(* CODESYS project Project_demo_2026_IOoff_v2_-_Codesys_SP20 (1)_RECOVERED_2026-05-21T15-52-03.project

Project tree, tasks and I/O mapping:
  Device : CODESYS Control Win V3 x64, CODESYS, version 3.5.20.40
    application Application
      libraries: Standard, 3.5.18.0 (System)
      task MainTask (cyclic, interval t#20ms, priority 1) calls PLC_PRG, SCADA_PRG, PRG_Loader, Order_generator
      function block Linear_Conveyor [SFC]: FB_Init, Receive_Workpiece_Data
      program PLC_PRG [CFC]
      data type Conv2Conv_bwd_T
      program Order_generator [ST]
      function block Cell [CFC]: FB_Init
      global variables GVL
      data type Conv2Conv_fwd_T
      data type Workpiece_T
      function block Machine_Conveyor [SFC]: FB_Init, Receive_Workpiece_Data, Inc_Next_Oper, Do_Change_Tool, Update_Tool, Copy_Next_Oper
      Symbols
      function block WarehouseIn_Conveyor [SFC]: Warehouse_Store_Piece, FB_Init, Warehouse_Rst_Piece, Receive_Workpiece_Data
      function block WarehouseOut_Conveyor [SFC]: FB_Init, Receive_Workpiece_Data, Warehouse_Req_Piece, Warehouse_Rst_Piece
      program SCADA_PRG [ST]
      data type Operation_T
      function block fb_Loader [ST]
      program PRG_Loader [ST]
      function block Transfer_Cell [CFC]: FB_Init
    Ethernet : Ethernet, CODESYS, version 4.2.0.0
      ModbusTCP_Slave_Device : ModbusTCP Server Device, CODESYS, version 4.4.0.0
          settings: UpdateableHolding = TRUE; DistinctBitAreas = TRUE; Coils Size = 8; Discrete Inputs Size = 8
          output S_sensor1 : BOOL  // Holding Registers.Holding Registers.Bit0
          output S_sensor2 : BOOL  // Holding Registers.Holding Registers.Bit1
          output S_sensor3 : BOOL  // Holding Registers.Holding Registers.Bit2
          output C1_stop : BOOL  // Holding Registers.Holding Registers.Bit0
          output C2_stop : BOOL  // Holding Registers.Holding Registers.Bit1
          output C3_stop : BOOL  // Holding Registers.Holding Registers.Bit2
          output Gate0 : BOOL  // Coils.Coils.Bit0
          output Gate1 : BOOL  // Coils.Coils.Bit1
          output Gate2 : BOOL  // Coils.Coils.Bit2
          unmapped channels: Holding Registers, Input Registers, Coils, Discrete Inputs
      Modbus_TCP_Master : Modbus TCP Client, CODESYS, version 4.4.0.0
          settings: AutoReconnect = TRUE
        Modbus_TCP_Slave : Modbus TCP Server, CODESYS, version 4.4.0.0
            settings: Unit-ID = 255; IPAddress = [127, 0, 0, 1]; Port = 5502; Channel 0.Function Code = 2; Channel 0.Read Offset = 16#0000; Channel 0.Read Length = 140; Channel 0.Write Offset = 0; Channel 0.Write Length = 0; Channel 0.Cycle Time = 100; Channel 1.Function Code = 15; Channel 1.Read Offset = 0; Channel 1.Read Length = 0; Channel 1.Write Offset = 16#0000; Channel 1.Write Length = 216; Channel 1.Cycle Time = 100; Channel 2.Function Code = 16; Channel 2.Read Offset = 0; Channel 2.Read Length = 0; Channel 2.Write Offset = 16#0000; Channel 2.Write Length = 15; Channel 2.Cycle Time = 100
            input  Application.GVL.In[0] : BOOL  // Channel 0.Channel 0.Bit0
            input  Application.GVL.In[1] : BOOL  // Channel 0.Channel 0.Bit1
            input  Application.GVL.In[2] : BOOL  // Channel 0.Channel 0.Bit2
            input  Application.GVL.In[3] : BOOL  // Channel 0.Channel 0.Bit3
            input  Application.GVL.In[4] : BOOL  // Channel 0.Channel 0.Bit4
            input  Application.GVL.In[5] : BOOL  // Channel 0.Channel 0.Bit5
            input  Application.GVL.In[6] : BOOL  // Channel 0.Channel 0.Bit6
            input  Application.GVL.In[7] : BOOL  // Channel 0.Channel 0.Bit7
            input  Application.GVL.In[8] : BOOL  // Channel 0.Channel 0.Bit0
            input  Application.GVL.In[9] : BOOL  // Channel 0.Channel 0.Bit1
            input  Application.GVL.In[10] : BOOL  // Channel 0.Channel 0.Bit2
            input  Application.GVL.In[11] : BOOL  // Channel 0.Channel 0.Bit3
            input  Application.GVL.In[12] : BOOL  // Channel 0.Channel 0.Bit4
            input  Application.GVL.In[13] : BOOL  // Channel 0.Channel 0.Bit5
            input  Application.GVL.In[14] : BOOL  // Channel 0.Channel 0.Bit6
            input  Application.GVL.In[15] : BOOL  // Channel 0.Channel 0.Bit7
            input  Application.GVL.In[16] : BOOL  // Channel 0.Channel 0.Bit0
            input  Application.GVL.In[17] : BOOL  // Channel 0.Channel 0.Bit1
            input  Application.GVL.In[18] : BOOL  // Channel 0.Channel 0.Bit2
            input  Application.GVL.In[19] : BOOL  // Channel 0.Channel 0.Bit3
            input  Application.GVL.In[20] : BOOL  // Channel 0.Channel 0.Bit4
            input  Application.GVL.In[21] : BOOL  // Channel 0.Channel 0.Bit5
            input  Application.GVL.In[22] : BOOL  // Channel 0.Channel 0.Bit6
            input  Application.GVL.In[23] : BOOL  // Channel 0.Channel 0.Bit7
            input  Application.GVL.In[24] : BOOL  // Channel 0.Channel 0.Bit0
            input  Application.GVL.In[25] : BOOL  // Channel 0.Channel 0.Bit1
            input  Application.GVL.In[26] : BOOL  // Channel 0.Channel 0.Bit2
            input  Application.GVL.In[27] : BOOL  // Channel 0.Channel 0.Bit3
            input  Application.GVL.In[28] : BOOL  // Channel 0.Channel 0.Bit4
            input  Application.GVL.In[29] : BOOL  // Channel 0.Channel 0.Bit5
            input  Application.GVL.In[30] : BOOL  // Channel 0.Channel 0.Bit6
            input  Application.GVL.In[31] : BOOL  // Channel 0.Channel 0.Bit7
            input  Application.GVL.In[32] : BOOL  // Channel 0.Channel 0.Bit0
            input  Application.GVL.In[33] : BOOL  // Channel 0.Channel 0.Bit1
            input  Application.GVL.In[34] : BOOL  // Channel 0.Channel 0.Bit2
            input  Application.GVL.In[35] : BOOL  // Channel 0.Channel 0.Bit3
            input  Application.GVL.In[36] : BOOL  // Channel 0.Channel 0.Bit4
            input  Application.GVL.In[37] : BOOL  // Channel 0.Channel 0.Bit5
            input  Application.GVL.In[38] : BOOL  // Channel 0.Channel 0.Bit6
            input  Application.GVL.In[39] : BOOL  // Channel 0.Channel 0.Bit7
            input  Application.GVL.In[40] : BOOL  // Channel 0.Channel 0.Bit0
            input  Application.GVL.In[41] : BOOL  // Channel 0.Channel 0.Bit1
            input  Application.GVL.In[42] : BOOL  // Channel 0.Channel 0.Bit2
            input  Application.GVL.In[43] : BOOL  // Channel 0.Channel 0.Bit3
            input  Application.GVL.In[44] : BOOL  // Channel 0.Channel 0.Bit4
            input  Application.GVL.In[45] : BOOL  // Channel 0.Channel 0.Bit5
            input  Application.GVL.In[46] : BOOL  // Channel 0.Channel 0.Bit6
            input  Application.GVL.In[47] : BOOL  // Channel 0.Channel 0.Bit7
            input  Application.GVL.In[48] : BOOL  // Channel 0.Channel 0.Bit0
            input  Application.GVL.In[49] : BOOL  // Channel 0.Channel 0.Bit1
            input  Application.GVL.In[50] : BOOL  // Channel 0.Channel 0.Bit2
            input  Application.GVL.In[51] : BOOL  // Channel 0.Channel 0.Bit3
            input  Application.GVL.In[52] : BOOL  // Channel 0.Channel 0.Bit4
            input  Application.GVL.In[53] : BOOL  // Channel 0.Channel 0.Bit5
            input  Application.GVL.In[54] : BOOL  // Channel 0.Channel 0.Bit6
            input  Application.GVL.In[55] : BOOL  // Channel 0.Channel 0.Bit7
            input  Application.GVL.In[56] : BOOL  // Channel 0.Channel 0.Bit0
            input  Application.GVL.In[57] : BOOL  // Channel 0.Channel 0.Bit1
            input  Application.GVL.In[58] : BOOL  // Channel 0.Channel 0.Bit2
            input  Application.GVL.In[59] : BOOL  // Channel 0.Channel 0.Bit3
            input  Application.GVL.In[60] : BOOL  // Channel 0.Channel 0.Bit4
            input  Application.GVL.In[61] : BOOL  // Channel 0.Channel 0.Bit5
            input  Application.GVL.In[62] : BOOL  // Channel 0.Channel 0.Bit6
            input  Application.GVL.In[63] : BOOL  // Channel 0.Channel 0.Bit7
            input  Application.GVL.In[64] : BOOL  // Channel 0.Channel 0.Bit0
            input  Application.GVL.In[65] : BOOL  // Channel 0.Channel 0.Bit1
            input  Application.GVL.In[66] : BOOL  // Channel 0.Channel 0.Bit2
            input  Application.GVL.In[67] : BOOL  // Channel 0.Channel 0.Bit3
            input  Application.GVL.In[68] : BOOL  // Channel 0.Channel 0.Bit4
            input  Application.GVL.In[69] : BOOL  // Channel 0.Channel 0.Bit5
            input  Application.GVL.In[70] : BOOL  // Channel 0.Channel 0.Bit6
            input  Application.GVL.In[71] : BOOL  // Channel 0.Channel 0.Bit7
            input  Application.GVL.In[72] : BOOL  // Channel 0.Channel 0.Bit0
            input  Application.GVL.In[73] : BOOL  // Channel 0.Channel 0.Bit1
            input  Application.GVL.In[74] : BOOL  // Channel 0.Channel 0.Bit2
            input  Application.GVL.In[75] : BOOL  // Channel 0.Channel 0.Bit3
            input  Application.GVL.In[76] : BOOL  // Channel 0.Channel 0.Bit4
            input  Application.GVL.In[77] : BOOL  // Channel 0.Channel 0.Bit5
            input  Application.GVL.In[78] : BOOL  // Channel 0.Channel 0.Bit6
            input  Application.GVL.In[79] : BOOL  // Channel 0.Channel 0.Bit7
            input  Application.GVL.In[80] : BOOL  // Channel 0.Channel 0.Bit0
            input  Application.GVL.In[81] : BOOL  // Channel 0.Channel 0.Bit1
            input  Application.GVL.In[82] : BOOL  // Channel 0.Channel 0.Bit2
            input  Application.GVL.In[83] : BOOL  // Channel 0.Channel 0.Bit3
            input  Application.GVL.In[84] : BOOL  // Channel 0.Channel 0.Bit4
            input  Application.GVL.In[85] : BOOL  // Channel 0.Channel 0.Bit5
            input  Application.GVL.In[86] : BOOL  // Channel 0.Channel 0.Bit6
            input  Application.GVL.In[87] : BOOL  // Channel 0.Channel 0.Bit7
            input  Application.GVL.In[88] : BOOL  // Channel 0.Channel 0.Bit0
            input  Application.GVL.In[89] : BOOL  // Channel 0.Channel 0.Bit1
            input  Application.GVL.In[90] : BOOL  // Channel 0.Channel 0.Bit2
            input  Application.GVL.In[91] : BOOL  // Channel 0.Channel 0.Bit3
            input  Application.GVL.In[92] : BOOL  // Channel 0.Channel 0.Bit4
            input  Application.GVL.In[93] : BOOL  // Channel 0.Channel 0.Bit5
            input  Application.GVL.In[94] : BOOL  // Channel 0.Channel 0.Bit6
            input  Application.GVL.In[95] : BOOL  // Channel 0.Channel 0.Bit7
            input  Application.GVL.In[96] : BOOL  // Channel 0.Channel 0.Bit0
            input  Application.GVL.In[97] : BOOL  // Channel 0.Channel 0.Bit1
            input  Application.GVL.In[98] : BOOL  // Channel 0.Channel 0.Bit2
            input  Application.GVL.In[99] : BOOL  // Channel 0.Channel 0.Bit3
            input  Application.GVL.In[100] : BOOL  // Channel 0.Channel 0.Bit4
            input  Application.GVL.In[101] : BOOL  // Channel 0.Channel 0.Bit5
            input  Application.GVL.In[102] : BOOL  // Channel 0.Channel 0.Bit6
            input  Application.GVL.In[103] : BOOL  // Channel 0.Channel 0.Bit7
            input  Application.GVL.In[104] : BOOL  // Channel 0.Channel 0.Bit0
            input  Application.GVL.In[105] : BOOL  // Channel 0.Channel 0.Bit1
            input  Application.GVL.In[106] : BOOL  // Channel 0.Channel 0.Bit2
            input  Application.GVL.In[107] : BOOL  // Channel 0.Channel 0.Bit3
            input  Application.GVL.In[108] : BOOL  // Channel 0.Channel 0.Bit4
            input  Application.GVL.In[109] : BOOL  // Channel 0.Channel 0.Bit5
            input  Application.GVL.In[110] : BOOL  // Channel 0.Channel 0.Bit6
            input  Application.GVL.In[111] : BOOL  // Channel 0.Channel 0.Bit7
            input  Application.GVL.In[112] : BOOL  // Channel 0.Channel 0.Bit0
            input  Application.GVL.In[113] : BOOL  // Channel 0.Channel 0.Bit1
            input  Application.GVL.In[114] : BOOL  // Channel 0.Channel 0.Bit2
            input  Application.GVL.In[115] : BOOL  // Channel 0.Channel 0.Bit3
            input  Application.GVL.In[116] : BOOL  // Channel 0.Channel 0.Bit4
            input  Application.GVL.In[117] : BOOL  // Channel 0.Channel 0.Bit5
            input  Application.GVL.In[118] : BOOL  // Channel 0.Channel 0.Bit6
            input  Application.GVL.In[119] : BOOL  // Channel 0.Channel 0.Bit7
            input  Application.GVL.In[120] : BOOL  // Channel 0.Channel 0.Bit0
            input  Application.GVL.In[121] : BOOL  // Channel 0.Channel 0.Bit1
            input  Application.GVL.In[122] : BOOL  // Channel 0.Channel 0.Bit2
            input  Application.GVL.In[123] : BOOL  // Channel 0.Channel 0.Bit3
            input  Application.GVL.In[124] : BOOL  // Channel 0.Channel 0.Bit4
            input  Application.GVL.In[125] : BOOL  // Channel 0.Channel 0.Bit5
            input  Application.GVL.In[126] : BOOL  // Channel 0.Channel 0.Bit6
            input  Application.GVL.In[127] : BOOL  // Channel 0.Channel 0.Bit7
            input  Application.GVL.In[128] : BOOL  // Channel 0.Channel 0.Bit0
            input  Application.GVL.In[129] : BOOL  // Channel 0.Channel 0.Bit1
            input  Application.GVL.In[130] : BOOL  // Channel 0.Channel 0.Bit2
            input  Application.GVL.In[131] : BOOL  // Channel 0.Channel 0.Bit3
            input  Application.GVL.In[132] : BOOL  // Channel 0.Channel 0.Bit4
            input  Application.GVL.In[133] : BOOL  // Channel 0.Channel 0.Bit5
            input  Application.GVL.In[134] : BOOL  // Channel 0.Channel 0.Bit6
            input  Application.GVL.In[135] : BOOL  // Channel 0.Channel 0.Bit7
            input  Application.GVL.In[136] : BOOL  // Channel 0.Channel 0.Bit0
            input  Application.GVL.In[137] : BOOL  // Channel 0.Channel 0.Bit1
            input  Application.GVL.In[138] : BOOL  // Channel 0.Channel 0.Bit2
            input  Application.GVL.In[139] : BOOL  // Channel 0.Channel 0.Bit3
            output Application.GVL.Out[0] : BOOL  // Channel 1.Channel 1.Bit0
            output Application.GVL.Out[1] : BOOL  // Channel 1.Channel 1.Bit1
            output Application.GVL.Out[2] : BOOL  // Channel 1.Channel 1.Bit2
            output Application.GVL.Out[3] : BOOL  // Channel 1.Channel 1.Bit3
            output Application.GVL.Out[4] : BOOL  // Channel 1.Channel 1.Bit4
            output Application.GVL.Out[5] : BOOL  // Channel 1.Channel 1.Bit5
            output Application.GVL.Out[6] : BOOL  // Channel 1.Channel 1.Bit6
            output Application.GVL.Out[7] : BOOL  // Channel 1.Channel 1.Bit7
            output Application.GVL.Out[8] : BOOL  // Channel 1.Channel 1.Bit0
            output Application.GVL.Out[9] : BOOL  // Channel 1.Channel 1.Bit1
            output Application.GVL.Out[10] : BOOL  // Channel 1.Channel 1.Bit2
            output Application.GVL.Out[11] : BOOL  // Channel 1.Channel 1.Bit3
            output Application.GVL.Out[12] : BOOL  // Channel 1.Channel 1.Bit4
            output Application.GVL.Out[13] : BOOL  // Channel 1.Channel 1.Bit5
            output Application.GVL.Out[14] : BOOL  // Channel 1.Channel 1.Bit6
            output Application.GVL.Out[15] : BOOL  // Channel 1.Channel 1.Bit7
            output Application.GVL.Out[16] : BOOL  // Channel 1.Channel 1.Bit0
            output Application.GVL.Out[17] : BOOL  // Channel 1.Channel 1.Bit1
            output Application.GVL.Out[18] : BOOL  // Channel 1.Channel 1.Bit2
            output Application.GVL.Out[19] : BOOL  // Channel 1.Channel 1.Bit3
            output Application.GVL.Out[20] : BOOL  // Channel 1.Channel 1.Bit4
            output Application.GVL.Out[21] : BOOL  // Channel 1.Channel 1.Bit5
            output Application.GVL.Out[22] : BOOL  // Channel 1.Channel 1.Bit6
            output Application.GVL.Out[23] : BOOL  // Channel 1.Channel 1.Bit7
            output Application.GVL.Out[24] : BOOL  // Channel 1.Channel 1.Bit0
            output Application.GVL.Out[25] : BOOL  // Channel 1.Channel 1.Bit1
            output Application.GVL.Out[26] : BOOL  // Channel 1.Channel 1.Bit2
            output Application.GVL.Out[27] : BOOL  // Channel 1.Channel 1.Bit3
            output Application.GVL.Out[28] : BOOL  // Channel 1.Channel 1.Bit4
            output Application.GVL.Out[29] : BOOL  // Channel 1.Channel 1.Bit5
            output Application.GVL.Out[30] : BOOL  // Channel 1.Channel 1.Bit6
            output Application.GVL.Out[31] : BOOL  // Channel 1.Channel 1.Bit7
            output Application.GVL.Out[32] : BOOL  // Channel 1.Channel 1.Bit0
            output Application.GVL.Out[33] : BOOL  // Channel 1.Channel 1.Bit1
            output Application.GVL.Out[34] : BOOL  // Channel 1.Channel 1.Bit2
            output Application.GVL.Out[35] : BOOL  // Channel 1.Channel 1.Bit3
            output Application.GVL.Out[36] : BOOL  // Channel 1.Channel 1.Bit4
            output Application.GVL.Out[37] : BOOL  // Channel 1.Channel 1.Bit5
            output Application.GVL.Out[38] : BOOL  // Channel 1.Channel 1.Bit6
            output Application.GVL.Out[39] : BOOL  // Channel 1.Channel 1.Bit7
            output Application.GVL.Out[40] : BOOL  // Channel 1.Channel 1.Bit0
            output Application.GVL.Out[41] : BOOL  // Channel 1.Channel 1.Bit1
            output Application.GVL.Out[42] : BOOL  // Channel 1.Channel 1.Bit2
            output Application.GVL.Out[43] : BOOL  // Channel 1.Channel 1.Bit3
            output Application.GVL.Out[44] : BOOL  // Channel 1.Channel 1.Bit4
            output Application.GVL.Out[45] : BOOL  // Channel 1.Channel 1.Bit5
            output Application.GVL.Out[46] : BOOL  // Channel 1.Channel 1.Bit6
            output Application.GVL.Out[47] : BOOL  // Channel 1.Channel 1.Bit7
            output Application.GVL.Out[48] : BOOL  // Channel 1.Channel 1.Bit0
            output Application.GVL.Out[49] : BOOL  // Channel 1.Channel 1.Bit1
            output Application.GVL.Out[50] : BOOL  // Channel 1.Channel 1.Bit2
            output Application.GVL.Out[51] : BOOL  // Channel 1.Channel 1.Bit3
            output Application.GVL.Out[52] : BOOL  // Channel 1.Channel 1.Bit4
            output Application.GVL.Out[53] : BOOL  // Channel 1.Channel 1.Bit5
            output Application.GVL.Out[54] : BOOL  // Channel 1.Channel 1.Bit6
            output Application.GVL.Out[55] : BOOL  // Channel 1.Channel 1.Bit7
            output Application.GVL.Out[56] : BOOL  // Channel 1.Channel 1.Bit0
            output Application.GVL.Out[57] : BOOL  // Channel 1.Channel 1.Bit1
            output Application.GVL.Out[58] : BOOL  // Channel 1.Channel 1.Bit2
            output Application.GVL.Out[59] : BOOL  // Channel 1.Channel 1.Bit3
            output Application.GVL.Out[60] : BOOL  // Channel 1.Channel 1.Bit4
            output Application.GVL.Out[61] : BOOL  // Channel 1.Channel 1.Bit5
            output Application.GVL.Out[62] : BOOL  // Channel 1.Channel 1.Bit6
            output Application.GVL.Out[63] : BOOL  // Channel 1.Channel 1.Bit7
            output Application.GVL.Out[64] : BOOL  // Channel 1.Channel 1.Bit0
            output Application.GVL.Out[65] : BOOL  // Channel 1.Channel 1.Bit1
            output Application.GVL.Out[66] : BOOL  // Channel 1.Channel 1.Bit2
            output Application.GVL.Out[67] : BOOL  // Channel 1.Channel 1.Bit3
            output Application.GVL.Out[68] : BOOL  // Channel 1.Channel 1.Bit4
            output Application.GVL.Out[69] : BOOL  // Channel 1.Channel 1.Bit5
            output Application.GVL.Out[70] : BOOL  // Channel 1.Channel 1.Bit6
            output Application.GVL.Out[71] : BOOL  // Channel 1.Channel 1.Bit7
            output Application.GVL.Out[72] : BOOL  // Channel 1.Channel 1.Bit0
            output Application.GVL.Out[73] : BOOL  // Channel 1.Channel 1.Bit1
            output Application.GVL.Out[74] : BOOL  // Channel 1.Channel 1.Bit2
            output Application.GVL.Out[75] : BOOL  // Channel 1.Channel 1.Bit3
            output Application.GVL.Out[76] : BOOL  // Channel 1.Channel 1.Bit4
            output Application.GVL.Out[77] : BOOL  // Channel 1.Channel 1.Bit5
            output Application.GVL.Out[78] : BOOL  // Channel 1.Channel 1.Bit6
            output Application.GVL.Out[79] : BOOL  // Channel 1.Channel 1.Bit7
            output Application.GVL.Out[80] : BOOL  // Channel 1.Channel 1.Bit0
            output Application.GVL.Out[81] : BOOL  // Channel 1.Channel 1.Bit1
            output Application.GVL.Out[82] : BOOL  // Channel 1.Channel 1.Bit2
            output Application.GVL.Out[83] : BOOL  // Channel 1.Channel 1.Bit3
            output Application.GVL.Out[84] : BOOL  // Channel 1.Channel 1.Bit4
            output Application.GVL.Out[85] : BOOL  // Channel 1.Channel 1.Bit5
            output Application.GVL.Out[86] : BOOL  // Channel 1.Channel 1.Bit6
            output Application.GVL.Out[87] : BOOL  // Channel 1.Channel 1.Bit7
            output Application.GVL.Out[88] : BOOL  // Channel 1.Channel 1.Bit0
            output Application.GVL.Out[89] : BOOL  // Channel 1.Channel 1.Bit1
            output Application.GVL.Out[90] : BOOL  // Channel 1.Channel 1.Bit2
            output Application.GVL.Out[91] : BOOL  // Channel 1.Channel 1.Bit3
            output Application.GVL.Out[92] : BOOL  // Channel 1.Channel 1.Bit4
            output Application.GVL.Out[93] : BOOL  // Channel 1.Channel 1.Bit5
            output Application.GVL.Out[94] : BOOL  // Channel 1.Channel 1.Bit6
            output Application.GVL.Out[95] : BOOL  // Channel 1.Channel 1.Bit7
            output Application.GVL.Out[96] : BOOL  // Channel 1.Channel 1.Bit0
            output Application.GVL.Out[97] : BOOL  // Channel 1.Channel 1.Bit1
            output Application.GVL.Out[98] : BOOL  // Channel 1.Channel 1.Bit2
            output Application.GVL.Out[99] : BOOL  // Channel 1.Channel 1.Bit3
            output Application.GVL.Out[100] : BOOL  // Channel 1.Channel 1.Bit4
            output Application.GVL.Out[101] : BOOL  // Channel 1.Channel 1.Bit5
            output Application.GVL.Out[102] : BOOL  // Channel 1.Channel 1.Bit6
            output Application.GVL.Out[103] : BOOL  // Channel 1.Channel 1.Bit7
            output Application.GVL.Out[104] : BOOL  // Channel 1.Channel 1.Bit0
            output Application.GVL.Out[105] : BOOL  // Channel 1.Channel 1.Bit1
            output Application.GVL.Out[106] : BOOL  // Channel 1.Channel 1.Bit2
            output Application.GVL.Out[107] : BOOL  // Channel 1.Channel 1.Bit3
            output Application.GVL.Out[108] : BOOL  // Channel 1.Channel 1.Bit4
            output Application.GVL.Out[109] : BOOL  // Channel 1.Channel 1.Bit5
            output Application.GVL.Out[110] : BOOL  // Channel 1.Channel 1.Bit6
            output Application.GVL.Out[111] : BOOL  // Channel 1.Channel 1.Bit7
            output Application.GVL.Out[112] : BOOL  // Channel 1.Channel 1.Bit0
            output Application.GVL.Out[113] : BOOL  // Channel 1.Channel 1.Bit1
            output Application.GVL.Out[114] : BOOL  // Channel 1.Channel 1.Bit2
            output Application.GVL.Out[115] : BOOL  // Channel 1.Channel 1.Bit3
            output Application.GVL.Out[116] : BOOL  // Channel 1.Channel 1.Bit4
            output Application.GVL.Out[117] : BOOL  // Channel 1.Channel 1.Bit5
            output Application.GVL.Out[118] : BOOL  // Channel 1.Channel 1.Bit6
            output Application.GVL.Out[119] : BOOL  // Channel 1.Channel 1.Bit7
            output Application.GVL.Out[120] : BOOL  // Channel 1.Channel 1.Bit0
            output Application.GVL.Out[121] : BOOL  // Channel 1.Channel 1.Bit1
            output Application.GVL.Out[122] : BOOL  // Channel 1.Channel 1.Bit2
            output Application.GVL.Out[123] : BOOL  // Channel 1.Channel 1.Bit3
            output Application.GVL.Out[124] : BOOL  // Channel 1.Channel 1.Bit4
            output Application.GVL.Out[125] : BOOL  // Channel 1.Channel 1.Bit5
            output Application.GVL.Out[126] : BOOL  // Channel 1.Channel 1.Bit6
            output Application.GVL.Out[127] : BOOL  // Channel 1.Channel 1.Bit7
            output Application.GVL.Out[128] : BOOL  // Channel 1.Channel 1.Bit0
            output Application.GVL.Out[129] : BOOL  // Channel 1.Channel 1.Bit1
            output Application.GVL.Out[130] : BOOL  // Channel 1.Channel 1.Bit2
            output Application.GVL.Out[131] : BOOL  // Channel 1.Channel 1.Bit3
            output Application.GVL.Out[132] : BOOL  // Channel 1.Channel 1.Bit4
            output Application.GVL.Out[133] : BOOL  // Channel 1.Channel 1.Bit5
            output Application.GVL.Out[134] : BOOL  // Channel 1.Channel 1.Bit6
            output Application.GVL.Out[135] : BOOL  // Channel 1.Channel 1.Bit7
            output Application.GVL.Out[136] : BOOL  // Channel 1.Channel 1.Bit0
            output Application.GVL.Out[137] : BOOL  // Channel 1.Channel 1.Bit1
            output Application.GVL.Out[138] : BOOL  // Channel 1.Channel 1.Bit2
            output Application.GVL.Out[139] : BOOL  // Channel 1.Channel 1.Bit3
            output Application.GVL.Out[140] : BOOL  // Channel 1.Channel 1.Bit4
            output Application.GVL.Out[141] : BOOL  // Channel 1.Channel 1.Bit5
            output Application.GVL.Out[142] : BOOL  // Channel 1.Channel 1.Bit6
            output Application.GVL.Out[143] : BOOL  // Channel 1.Channel 1.Bit7
            output Application.GVL.Out[144] : BOOL  // Channel 1.Channel 1.Bit0
            output Application.GVL.Out[145] : BOOL  // Channel 1.Channel 1.Bit1
            output Application.GVL.Out[146] : BOOL  // Channel 1.Channel 1.Bit2
            output Application.GVL.Out[147] : BOOL  // Channel 1.Channel 1.Bit3
            output Application.GVL.Out[148] : BOOL  // Channel 1.Channel 1.Bit4
            output Application.GVL.Out[149] : BOOL  // Channel 1.Channel 1.Bit5
            output Application.GVL.Out[150] : BOOL  // Channel 1.Channel 1.Bit6
            output Application.GVL.Out[151] : BOOL  // Channel 1.Channel 1.Bit7
            output Application.GVL.Out[152] : BOOL  // Channel 1.Channel 1.Bit0
            output Application.GVL.Out[153] : BOOL  // Channel 1.Channel 1.Bit1
            output Application.GVL.Out[154] : BOOL  // Channel 1.Channel 1.Bit2
            output Application.GVL.Out[155] : BOOL  // Channel 1.Channel 1.Bit3
            output Application.GVL.Out[156] : BOOL  // Channel 1.Channel 1.Bit4
            output Application.GVL.Out[157] : BOOL  // Channel 1.Channel 1.Bit5
            output Application.GVL.Out[158] : BOOL  // Channel 1.Channel 1.Bit6
            output Application.GVL.Out[159] : BOOL  // Channel 1.Channel 1.Bit7
            output Application.GVL.Out[160] : BOOL  // Channel 1.Channel 1.Bit0
            output Application.GVL.Out[161] : BOOL  // Channel 1.Channel 1.Bit1
            output Application.GVL.Out[162] : BOOL  // Channel 1.Channel 1.Bit2
            output Application.GVL.Out[163] : BOOL  // Channel 1.Channel 1.Bit3
            output Application.GVL.Out[164] : BOOL  // Channel 1.Channel 1.Bit4
            output Application.GVL.Out[165] : BOOL  // Channel 1.Channel 1.Bit5
            output Application.GVL.Out[166] : BOOL  // Channel 1.Channel 1.Bit6
            output Application.GVL.Out[167] : BOOL  // Channel 1.Channel 1.Bit7
            output Application.GVL.Out[168] : BOOL  // Channel 1.Channel 1.Bit0
            output Application.GVL.Out[169] : BOOL  // Channel 1.Channel 1.Bit1
            output Application.GVL.Out[170] : BOOL  // Channel 1.Channel 1.Bit2
            output Application.GVL.Out[171] : BOOL  // Channel 1.Channel 1.Bit3
            output Application.GVL.Out[172] : BOOL  // Channel 1.Channel 1.Bit4
            output Application.GVL.Out[173] : BOOL  // Channel 1.Channel 1.Bit5
            output Application.GVL.Out[174] : BOOL  // Channel 1.Channel 1.Bit6
            output Application.GVL.Out[175] : BOOL  // Channel 1.Channel 1.Bit7
            output Application.GVL.Out[176] : BOOL  // Channel 1.Channel 1.Bit0
            output Application.GVL.Out[177] : BOOL  // Channel 1.Channel 1.Bit1
            output Application.GVL.Out[178] : BOOL  // Channel 1.Channel 1.Bit2
            output Application.GVL.Out[179] : BOOL  // Channel 1.Channel 1.Bit3
            output Application.GVL.Out[180] : BOOL  // Channel 1.Channel 1.Bit4
            output Application.GVL.Out[181] : BOOL  // Channel 1.Channel 1.Bit5
            output Application.GVL.Out[182] : BOOL  // Channel 1.Channel 1.Bit6
            output Application.GVL.Out[183] : BOOL  // Channel 1.Channel 1.Bit7
            output Application.GVL.Out[184] : BOOL  // Channel 1.Channel 1.Bit0
            output Application.GVL.Out[185] : BOOL  // Channel 1.Channel 1.Bit1
            output Application.GVL.Out[186] : BOOL  // Channel 1.Channel 1.Bit2
            output Application.GVL.Out[187] : BOOL  // Channel 1.Channel 1.Bit3
            output Application.GVL.Out[188] : BOOL  // Channel 1.Channel 1.Bit4
            output Application.GVL.Out[189] : BOOL  // Channel 1.Channel 1.Bit5
            output Application.GVL.Out[190] : BOOL  // Channel 1.Channel 1.Bit6
            output Application.GVL.Out[191] : BOOL  // Channel 1.Channel 1.Bit7
            output Application.GVL.Out[192] : BOOL  // Channel 1.Channel 1.Bit0
            output Application.GVL.Out[193] : BOOL  // Channel 1.Channel 1.Bit1
            output Application.GVL.Out[194] : BOOL  // Channel 1.Channel 1.Bit2
            output Application.GVL.Out[195] : BOOL  // Channel 1.Channel 1.Bit3
            output Application.GVL.Out[196] : BOOL  // Channel 1.Channel 1.Bit4
            output Application.GVL.Out[197] : BOOL  // Channel 1.Channel 1.Bit5
            output Application.GVL.Out[198] : BOOL  // Channel 1.Channel 1.Bit6
            output Application.GVL.Out[199] : BOOL  // Channel 1.Channel 1.Bit7
            output Application.GVL.Out[200] : BOOL  // Channel 1.Channel 1.Bit0
            output Application.GVL.Out[201] : BOOL  // Channel 1.Channel 1.Bit1
            output Application.GVL.Out[202] : BOOL  // Channel 1.Channel 1.Bit2
            output Application.GVL.Out[203] : BOOL  // Channel 1.Channel 1.Bit3
            output Application.GVL.Out[204] : BOOL  // Channel 1.Channel 1.Bit4
            output Application.GVL.Out[205] : BOOL  // Channel 1.Channel 1.Bit5
            output Application.GVL.Out[206] : BOOL  // Channel 1.Channel 1.Bit6
            output Application.GVL.Out[207] : BOOL  // Channel 1.Channel 1.Bit7
            output Application.GVL.Out[208] : BOOL  // Channel 1.Channel 1.Bit0
            output Application.GVL.Out[209] : BOOL  // Channel 1.Channel 1.Bit1
            output Application.GVL.Out[210] : BOOL  // Channel 1.Channel 1.Bit2
            output Application.GVL.Out[211] : BOOL  // Channel 1.Channel 1.Bit3
            output Application.GVL.Out[212] : BOOL  // Channel 1.Channel 1.Bit4
            output Application.GVL.Out[213] : BOOL  // Channel 1.Channel 1.Bit5
            output Application.GVL.Out[214] : BOOL  // Channel 1.Channel 1.Bit6
            output Application.GVL.Out[215] : BOOL  // Channel 1.Channel 1.Bit7
            output Application.GVL.Reg[0] : WORD  // Channel 2.Channel 2
            output Application.GVL.Reg[1] : WORD  // Channel 2.Channel 2
            output Application.GVL.Reg[2] : WORD  // Channel 2.Channel 2
            output Application.GVL.Reg[3] : WORD  // Channel 2.Channel 2
            output Application.GVL.Reg[4] : WORD  // Channel 2.Channel 2
            output Application.GVL.Reg[5] : WORD  // Channel 2.Channel 2
            output Application.GVL.Reg[6] : WORD  // Channel 2.Channel 2
            output Application.GVL.Reg[7] : WORD  // Channel 2.Channel 2
            output Application.GVL.Reg[8] : WORD  // Channel 2.Channel 2
            output Application.GVL.Reg[9] : WORD  // Channel 2.Channel 2
            output Application.GVL.Reg[10] : WORD  // Channel 2.Channel 2
            output Application.GVL.Reg[11] : WORD  // Channel 2.Channel 2
            output Application.GVL.Reg[12] : WORD  // Channel 2.Channel 2
            output Application.GVL.Reg[13] : WORD  // Channel 2.Channel 2
            output Application.GVL.Reg[14] : WORD  // Channel 2.Channel 2
            unmapped channels: Channel 0, Channel 1, Channel 2
*)

// Device/Application/Conv2Conv_bwd_T
TYPE Conv2Conv_bwd_T :
STRUCT
		free_cmd: BOOL;
END_STRUCT
END_TYPE

// Device/Application/Conv2Conv_fwd_T
TYPE Conv2Conv_fwd_T :
STRUCT
		recv_cmd: BOOL;
		Workpiece: Workpiece_T;
END_STRUCT
END_TYPE

// Device/Application/Workpiece_T
TYPE Workpiece_T :
STRUCT
	InitPiece: INT;
	Operations: ARRAY [0 .. 10] OF Operation_T;
	Next_Operation: INT;
	Last_Operation: INT;
END_STRUCT
END_TYPE

// Device/Application/Operation_T
TYPE Operation_T :
STRUCT
	Cell: INT;
	Machine: INT;
	Tool: INT;
	OpTime: TIME;
END_STRUCT
END_TYPE

// Device/Application/GVL
{attribute 'qualified_only'}
VAR_GLOBAL
	In:  ARRAY [0 .. 139] OF BOOL;
	Out: ARRAY [0 .. 215] OF BOOL;
	Reg: ARRAY [0 .. 14] OF UINT;
	
	Cell_1_Top_Order:  Conv2conv_fwd_T;
	Cell_1_Top_Status: Conv2conv_bwd_T;
	
	Cell_2_Top_Order:  Conv2conv_fwd_T;
	Cell_2_Top_Status: Conv2conv_bwd_T;
	
	// Add to existing GVL VAR_GLOBAL block:

	// Cells 3 & 4 handshakes (já tens no PLC_PRG, move-os para GVL para acesso OPC-UA)
	Cell_3_Top_Order:  Conv2Conv_fwd_T;
	Cell_3_Top_Status: Conv2Conv_bwd_T;
	Cell_4_Top_Order:  Conv2Conv_fwd_T;
	Cell_4_Top_Status: Conv2Conv_bwd_T;
	
	// Transfer cell
	Transfer_Order  : Conv2Conv_fwd_T;
	Transfer_Status : Conv2Conv_bwd_T;

// Loader / Unloader / Return
g_Loader_Wood_Qty:    INT;
g_Loader_Metal_Qty:   INT;
g_Loader_Exec:        BOOL;

g_Unloader_PieceType: STRING;
g_Unloader_Qty:       INT;
g_Unloader_Exec:      BOOL;

g_Return_PieceID:     INT;
g_Return_Exec:        BOOL;

// Warehouse counters (PLC increments/decrements on load/unload events)
g_W1_Count: INT;
g_W2_Count: INT;

g_Loader_Status: INT; // 0 = IDLE, 1 = LOADING, 2 = DONE, 3 = ERROR
END_VAR

// Device/Application/PLC_PRG
PROGRAM PLC_PRG
VAR
	Cell_1: Cell(
        11, 28, 5,     			// Wout_I, Wout_Q, Wout_R
        30, 70, 1, 1, 2, 3,		// M1_I, M1_Q, M1_InitTool, M1_Tool1, M1_Tool2, M1_Tool3
        36, 80,					// T1_I, T1_Q
        37, 82, 1, 1, 2, 3,    	// M2_I, M2_Q, M2_InitTool, M2_Tool1, M2_Tool2, M2_Tool3
        43, 92,        			// T2_I, T2_Q
        44, 94, 8, 8, 9, 11,    // M3_I, M3_Q, M3_InitTool, M3_Tool1, M3_Tool2, M3_Tool3
        21, 48, 0      			// Win_I, Win_Q, Win_R
	);
	
	Cell_2: Cell(
        12, 30, 6,     			// Wout_I, Wout_Q, Wout_R
        50, 104, 1, 1, 2, 3,    // M1_I, M1_Q, M1_InitTool, M1_Tool1, M1_Tool2, M1_Tool3
        56, 114,        		// T1_I, T1_Q
        57, 116, 1, 1, 2, 3,    // M2_I, M2_Q, M2_InitTool, M2_Tool1, M2_Tool2, M2_Tool3
        63, 126,        		// T2_I, T2_Q
        64, 128, 8, 8, 9, 10,   // M3_I, M3_Q, M3_InitTool, M3_Tool1, M3_Tool2, M3_Tool3
        22, 51, 0      			// Win_I, Win_Q, Win_R
	);
	
	Cell_3: Cell(
        13, 32, 7,     			// Wout_I, Wout_Q, Wout_R
        70, 138, 4, 4, 5, 6,    // M1_I, M1_Q, M1_InitTool, M1_Tool1, M1_Tool2, M1_Tool3
        76, 148,        		// T1_I, T1_Q
        77, 150, 4, 4, 5, 6,    // M2_I, M2_Q, M2_InitTool, M2_Tool1, M2_Tool2, M2_Tool3
        83, 160,        		// T2_I, T2_Q
        84, 162, 8, 8, 9, 11,   // M3_I, M3_Q, M3_InitTool, M3_Tool1, M3_Tool2, M3_Tool3
        23, 54, 0      			// Win_I, Win_Q, Win_R
	);
	
	Cell_4: Cell(
        14, 34, 8,     			 // Wout_I, Wout_Q, Wout_R
        90, 172, 4, 4, 5, 6,     // M1_I, M1_Q, M1_InitTool, M1_Tool1, M1_Tool2, M1_Tool3
        96, 182,        		 // T1_I, T1_Q
        97, 184, 4, 4, 5, 6,     // M2_I, M2_Q, M2_InitTool, M2_Tool1, M2_Tool2, M2_Tool3
        103, 194,        		 // T2_I, T2_Q
        104, 196, 8, 8, 9, 10,   // M3_I, M3_Q, M3_InitTool, M3_Tool1, M3_Tool2, M3_Tool3
        24, 57, 0      			 // Win_I, Win_Q, Win_R
	);
	
	Transfer: Transfer_Cell(
		20, 45, 14,				// Wout_I, Wout_Q, Wout_R
		29, 67,        		    // T1_I, T1_Q
		28, 65,        		    // T2_I, T2_Q
		27, 63,        		    // T3_I, T3_Q
		26, 61,        		    // T4_I, T4_Q
		25, 59,        		    // T5_I, T5_Q
		10, 24, 0      			// Win_I, Win_Q, Win_R
	);
END_VAR

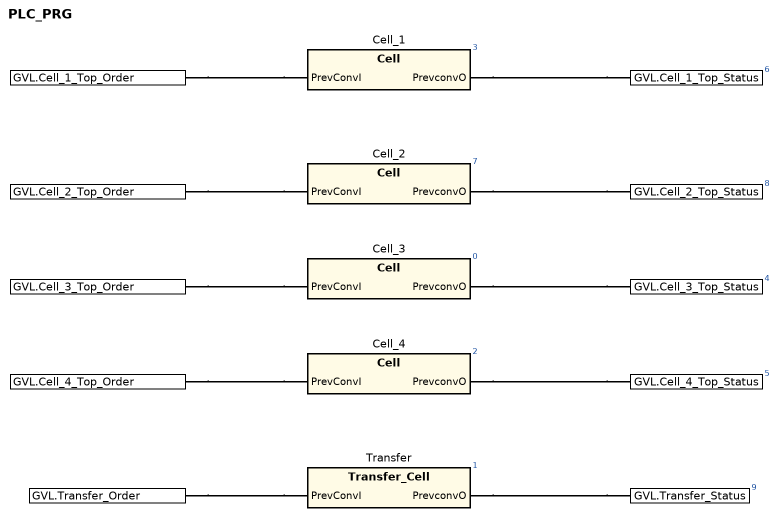
Cell_3(PrevConvI := GVL.Cell_3_Top_Order); // Cell
Transfer(PrevConvI := GVL.Transfer_Order); // Transfer_Cell
Cell_4(PrevConvI := GVL.Cell_4_Top_Order); // Cell
Cell_1(PrevConvI := GVL.Cell_1_Top_Order); // Cell
GVL.Cell_3_Top_Status := Cell_3.PrevconvO;
GVL.Cell_4_Top_Status := Cell_4.PrevconvO;
GVL.Cell_1_Top_Status := Cell_1.PrevconvO;
Cell_2(PrevConvI := GVL.Cell_2_Top_Order); // Cell
GVL.Cell_2_Top_Status := Cell_2.PrevconvO;
GVL.Transfer_Status := Transfer.PrevconvO;

END_PROGRAM

// Device/Application/Cell
FUNCTION_BLOCK Cell
VAR_INPUT
	PrevConvI: Conv2Conv_fwd_T;
	M1_InitTool : INT;
	M1_Tool1 : INT;
    M1_Tool2 : INT;
    M1_Tool3 : INT;
	M2_InitTool : INT;
	M2_Tool1 : INT;
    M2_Tool2 : INT;
    M2_Tool3 : INT;
	M3_InitTool : INT;
	M3_Tool1 : INT;
    M3_Tool2 : INT;
    M3_Tool3 : INT;
END_VAR
VAR_OUTPUT
	PrevconvO: Conv2Conv_bwd_T;
END_VAR
VAR
	Wout : WarehouseOut_Conveyor(0, 0, 0);
	M1   : Machine_Conveyor(1, 0, 0, 0, 0, 0, 0, 0);
	T1   : Linear_Conveyor(0, 0, 0);
	M2   : Machine_Conveyor(2, 0, 0, 0, 0, 0, 0, 0);
	T2	 : Linear_Conveyor(0, 0, 0);
	M3   : Machine_Conveyor(3, 0, 0, 0, 0, 0, 0, 0);
	Win  : WarehouseIn_Conveyor(0, 0, 0);
END_VAR

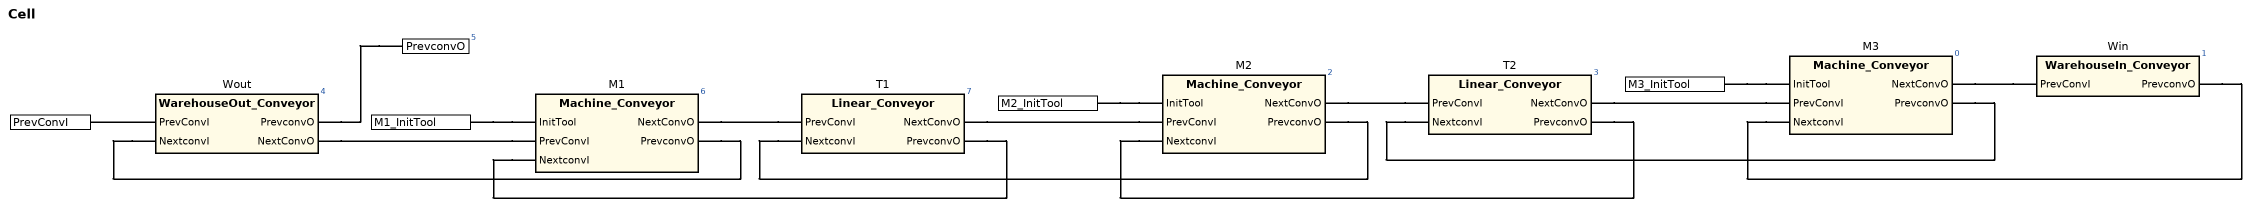
M3(InitTool := M3_InitTool, PrevConvI := T2.NextConvO, NextconvI := Win.PrevconvO); // Machine_Conveyor
Win(PrevConvI := M3.NextConvO); // WarehouseIn_Conveyor
M2(InitTool := M2_InitTool, PrevConvI := T1.NextConvO, NextconvI := T2.PrevconvO); // Machine_Conveyor
T2(PrevConvI := M2.NextConvO, NextconvI := M3.PrevconvO); // Linear_Conveyor
Wout(PrevConvI := PrevConvI, NextconvI := M1.PrevconvO); // WarehouseOut_Conveyor
PrevconvO := Wout.PrevconvO;
M1(InitTool := M1_InitTool, PrevConvI := Wout.NextConvO, NextconvI := T1.PrevconvO); // Machine_Conveyor
T1(PrevConvI := M1.NextConvO, NextconvI := M2.PrevconvO); // Linear_Conveyor

//FB_Init is always available implicitly and it is used primarily for initialization.
//The return value is not evaluated. For a specific influence, you can also declare the
//methods explicitly and provide additional code there with the standard initialization
//code. You can evaluate the return value.
METHOD FB_Init: BOOL
VAR_INPUT
    bInitRetains: BOOL; // TRUE: the retain variables are initialized (reset warm / reset cold)
    bInCopyCode: BOOL;  // TRUE: the instance will be copied to the copy code afterward (online change)   
	Wout_I_ : INT; Wout_Q_ : INT; Wout_R_ : INT;
	M1_I_ : INT; M1_Q_ : INT; M1_InitTool_ : INT; M1_Tool1_ : INT; M1_Tool2_ : INT; M1_Tool3_ : INT;
	T1_I_ : INT; T1_Q_ : INT;
	M2_I_ : INT; M2_Q_ : INT; M2_InitTool_ : INT; M2_Tool1_ : INT; M2_Tool2_ : INT; M2_Tool3_ : INT;
	T2_I_ : INT; T2_Q_ : INT;
	M3_I_ : INT; M3_Q_ : INT; M3_InitTool_ : INT; M3_Tool1_ : INT; M3_Tool2_ : INT; M3_Tool3_ : INT;
	Win_I_ : INT; Win_Q_ : INT; Win_R_ : INT;
END_VAR
	(* Codesys seems to be calling the FB_init methods in the inverse order,
	 * so we call them here again with the correct values
	 *)
	Wout.FB_Init(FALSE, FALSE, Wout_I_, Wout_Q_, Wout_R_);
	M1.FB_Init(FALSE, FALSE, 1, M1_InitTool_, M1_Tool1_, M1_Tool2_, M1_Tool3_, M1_I_, M1_Q_, 0);
	T1.FB_Init(FALSE, FALSE, T1_I_, T1_Q_, 0);
	M2.FB_Init(FALSE, FALSE, 2, M2_InitTool_, M2_Tool1_, M2_Tool2_, M2_Tool3_, M2_I_, M2_Q_, 0);
	T2.FB_Init(FALSE, FALSE, T2_I_, T2_Q_, 0);
	M3.FB_Init(FALSE, FALSE, 3, M3_InitTool_, M3_Tool1_, M3_Tool2_, M3_Tool3_, M3_I_, M3_Q_, 0);
	Win.FB_Init(FALSE, FALSE, Win_I_, Win_Q_, Win_R_);
END_METHOD

END_FUNCTION_BLOCK

// Device/Application/Machine_Conveyor
FUNCTION_BLOCK Machine_Conveyor
VAR_INPUT
	MachineID: INT;
	InitTool: INT;
	NextconvI: Conv2Conv_bwd_T;
	PrevConvI: Conv2Conv_fwd_T;
END_VAR
VAR_OUTPUT
	PrevconvO: Conv2Conv_bwd_T;
	NextConvO: Conv2Conv_fwd_T;
END_VAR
VAR
	Ioff: INT;
	Qoff: INT;
	Tool: INT;
	Tool1: INT;
	Tool2: INT;
	Tool3: INT;
	NextOper: Operation_T;
	ToolSensorReady : BOOL;
	ToolChanged : BOOL;
END_VAR

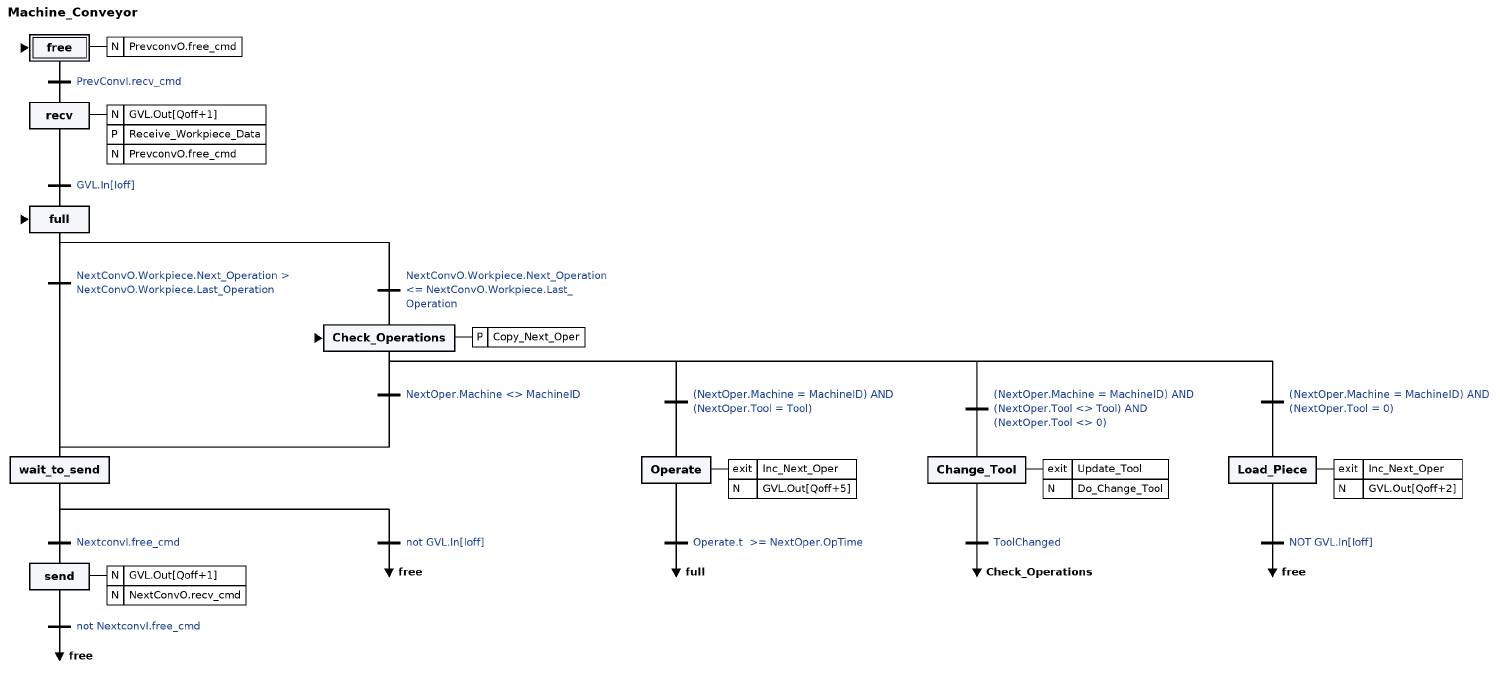
INITIAL_STEP free:
    PrevconvO.free_cmd(N);
END_STEP
TRANSITION FROM free TO recv
    := PrevConvI.recv_cmd;
END_TRANSITION
STEP recv:
    GVL.Out[Qoff+1](N);
    Receive_Workpiece_Data(P);
    PrevconvO.free_cmd(N);
END_STEP
TRANSITION FROM recv TO full
    := GVL.In[Ioff];
END_TRANSITION
STEP full:
END_STEP
TRANSITION FROM full TO wait_to_send
    := NextConvO.Workpiece.Next_Operation > NextConvO.Workpiece.Last_Operation;
END_TRANSITION
TRANSITION FROM full TO Check_Operations
    := NextConvO.Workpiece.Next_Operation <= NextConvO.Workpiece.Last_Operation;
END_TRANSITION
STEP Check_Operations:
    Copy_Next_Oper(P);
END_STEP
TRANSITION FROM Check_Operations TO wait_to_send
    := NextOper.Machine <> MachineID;
END_TRANSITION
TRANSITION FROM Check_Operations TO Operate
    := (NextOper.Machine = MachineID) AND (NextOper.Tool = Tool);
END_TRANSITION
STEP Operate:
    Inc_Next_Oper(P0);  // exit action
    GVL.Out[Qoff+5](N);
END_STEP
TRANSITION FROM Operate TO full
    := Operate.t >= NextOper.OpTime;
END_TRANSITION
TRANSITION FROM Check_Operations TO Change_Tool
    := (NextOper.Machine = MachineID) AND (NextOper.Tool <> Tool) AND (NextOper.Tool <> 0);
END_TRANSITION
STEP Change_Tool:
    Update_Tool(P0);  // exit action
    Do_Change_Tool(N);
END_STEP
TRANSITION FROM Change_Tool TO Check_Operations
    := ToolChanged;
END_TRANSITION
TRANSITION FROM Check_Operations TO Load_Piece
    := (NextOper.Machine = MachineID) AND (NextOper.Tool = 0);
END_TRANSITION
STEP Load_Piece:
    Inc_Next_Oper(P0);  // exit action
    GVL.Out[Qoff+2](N);
END_STEP
TRANSITION FROM Load_Piece TO free
    := NOT GVL.In[Ioff];
END_TRANSITION
STEP wait_to_send:
END_STEP
TRANSITION FROM wait_to_send TO send
    := NextconvI.free_cmd;
END_TRANSITION
TRANSITION FROM wait_to_send TO free
    := not GVL.In[Ioff];
END_TRANSITION
STEP send:
    GVL.Out[Qoff+1](N);
    NextConvO.recv_cmd(N);
END_STEP
TRANSITION FROM send TO free
    := not NextconvI.free_cmd;
END_TRANSITION

//FB_Init is always available implicitly and it is used primarily for initialization.
//The return value is not evaluated. For a specific influence, you can also declare the
//methods explicitly and provide additional code there with the standard initialization
//code. You can evaluate the return value.
METHOD FB_Init: BOOL
VAR_INPUT
    bInitRetains: BOOL; // TRUE: the retain variables are initialized (reset warm / reset cold)
    bInCopyCode: BOOL;  // TRUE: the instance will be copied to the copy code afterward (online change)   
	MachineID_: INT;
	Tool_ : INT;
	Tool1_: INT;
	Tool2_: INT;
 	Tool3_: INT;
	Ioff_	: INT;
	Qoff_	: INT;
	Roff_	: INT;	
END_VAR
	MachineID := MachineID_;
	Tool := Tool_;
	Tool1 := Tool1_;
	Tool2 := Tool2_;
	Tool3 := Tool3_;
	Ioff := Ioff_;
	Qoff := Qoff_;
	//Roff := Roff_;
END_METHOD

ACTION Receive_Workpiece_Data:
NextConvO.Workpiece := PrevConvI.Workpiece;
END_ACTION

ACTION Inc_Next_Oper:
NextConvO.Workpiece.Next_Operation := NextConvO.Workpiece.Next_Operation + 1;
END_ACTION

ACTION Do_Change_Tool:
IF Tool = Tool1 THEN
    IF NextOper.Tool = Tool2 THEN
        GVL.Out[Qoff + 3] := TRUE; // Rotate -
    ELSIF NextOper.Tool = Tool3 THEN
        GVL.Out[Qoff + 4] := TRUE; // Rotate +
    END_IF;

ELSIF Tool = Tool2 THEN
    IF NextOper.Tool = Tool3 THEN
        GVL.Out[Qoff + 3] := TRUE;
    ELSIF NextOper.Tool = Tool1 THEN
        GVL.Out[Qoff + 4] := TRUE;
    END_IF;

ELSIF Tool = Tool3 THEN
    IF NextOper.Tool = Tool1 THEN
        GVL.Out[Qoff + 3] := TRUE;
    ELSIF NextOper.Tool = Tool2 THEN
        GVL.Out[Qoff + 4] := TRUE;
    END_IF;
END_IF;

IF NOT GVL.In[Ioff + 1] THEN
    ToolSensorReady := TRUE;
END_IF;

IF ToolSensorReady AND GVL.In[Ioff + 1] THEN
    ToolChanged := TRUE;
END_IF;
END_ACTION

ACTION Update_Tool:
Tool := NextOper.Tool;

GVL.Out[Qoff + 3] := FALSE; // Rotate -
GVL.Out[Qoff + 4] := FALSE; // Rotate +

ToolSensorReady := FALSE;
ToolChanged := FALSE;
END_ACTION

ACTION Copy_Next_Oper:
NextOper := NextConvO.Workpiece.Operations[NextConvO.Workpiece.Next_Operation];
END_ACTION

END_FUNCTION_BLOCK

// Device/Application/Linear_Conveyor
FUNCTION_BLOCK Linear_Conveyor
VAR_INPUT
	NextconvI: Conv2Conv_bwd_T;
	PrevConvI: Conv2Conv_fwd_T;
END_VAR
VAR_OUTPUT
	PrevconvO: Conv2Conv_bwd_T;
	NextConvO: Conv2Conv_fwd_T;
END_VAR
VAR
	Ioff: INT;
	Qoff: INT;
	x: INT;
END_VAR

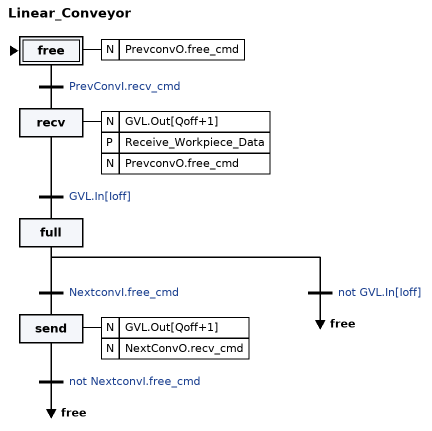
INITIAL_STEP free:
    PrevconvO.free_cmd(N);
END_STEP
TRANSITION FROM free TO recv
    := PrevConvI.recv_cmd;
END_TRANSITION
STEP recv:
    GVL.Out[Qoff+1](N);
    Receive_Workpiece_Data(P);
    PrevconvO.free_cmd(N);
END_STEP
TRANSITION FROM recv TO full
    := GVL.In[Ioff];
END_TRANSITION
STEP full:
END_STEP
TRANSITION FROM full TO send
    := NextconvI.free_cmd;
END_TRANSITION
TRANSITION FROM full TO free
    := not GVL.In[Ioff];
END_TRANSITION
STEP send:
    GVL.Out[Qoff+1](N);
    NextConvO.recv_cmd(N);
END_STEP
TRANSITION FROM send TO free
    := not NextconvI.free_cmd;
END_TRANSITION

//FB_Init is always available implicitly and it is used primarily for initialization.
//The return value is not evaluated. For a specific influence, you can also declare the
//methods explicitly and provide additional code there with the standard initialization
//code. You can evaluate the return value.
METHOD FB_Init: BOOL
VAR_INPUT
    bInitRetains: BOOL; // TRUE: the retain variables are initialized (reset warm / reset cold)
    bInCopyCode: BOOL;  // TRUE: the instance will be copied to the copy code afterward (online change)   
	Ioff_	: INT;
	Qoff_	: INT;
	Roff_	: INT;	
END_VAR
	Ioff := Ioff_;
	Qoff := Qoff_;
	//Roff := Roff_;
	x := x + 1;
END_METHOD

ACTION Receive_Workpiece_Data:
NextConvO.Workpiece := PrevConvI.Workpiece;
END_ACTION

END_FUNCTION_BLOCK

// Device/Application/WarehouseOut_Conveyor
FUNCTION_BLOCK WarehouseOut_Conveyor
VAR_INPUT
	NextconvI: Conv2Conv_bwd_T;
	PrevConvI: Conv2Conv_fwd_T;
END_VAR
VAR_OUTPUT
	NextConvO: Conv2Conv_fwd_T;
	PrevconvO: Conv2Conv_bwd_T;
END_VAR
VAR
	Ioff: INT;
	Qoff: INT;
	Roff: INT;
END_VAR

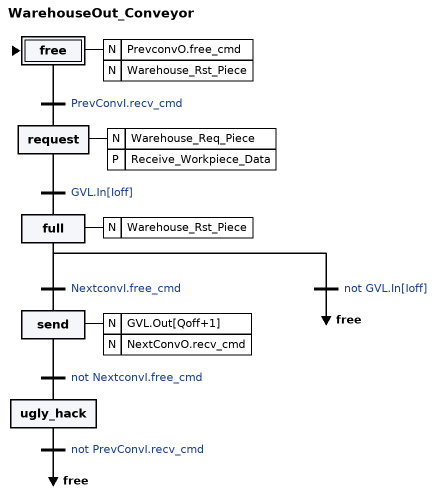
INITIAL_STEP free:
    PrevconvO.free_cmd(N);
    Warehouse_Rst_Piece(N);
END_STEP
TRANSITION FROM free TO request
    := PrevConvI.recv_cmd;
END_TRANSITION
STEP request:
    Warehouse_Req_Piece(N);
    Receive_Workpiece_Data(P);
END_STEP
TRANSITION FROM request TO full
    := GVL.In[Ioff];
END_TRANSITION
STEP full:
    Warehouse_Rst_Piece(N);
END_STEP
TRANSITION FROM full TO send
    := NextconvI.free_cmd;
END_TRANSITION
TRANSITION FROM full TO free
    := not GVL.In[Ioff];
END_TRANSITION
STEP send:
    GVL.Out[Qoff+1](N);
    NextConvO.recv_cmd(N);
END_STEP
TRANSITION FROM send TO ugly_hack
    := not NextconvI.free_cmd;
END_TRANSITION
STEP ugly_hack:
END_STEP
TRANSITION FROM ugly_hack TO free
    := not PrevConvI.recv_cmd;
END_TRANSITION

//FB_Init is always available implicitly and it is used primarily for initialization.
//The return value is not evaluated. For a specific influence, you can also declare the
//methods explicitly and provide additional code there with the standard initialization
//code. You can evaluate the return value.
METHOD FB_Init: BOOL
VAR_INPUT
    bInitRetains: BOOL; // TRUE: the retain variables are initialized (reset warm / reset cold)
    bInCopyCode: BOOL;  // TRUE: the instance will be copied to the copy code afterward (online change)   
	Ioff_	: INT;
	Qoff_	: INT;
	Roff_	: INT;	
END_VAR
	Ioff := Ioff_;
	Qoff := Qoff_;
	Roff := Roff_;
END_METHOD

ACTION Receive_Workpiece_Data:
NextConvO.Workpiece := PrevConvI.Workpiece;
PrevConvI.recv_cmd := false;
END_ACTION

ACTION Warehouse_Req_Piece:
GVL.Reg[Roff] := TO_UINT(PrevConvI.Workpiece.InitPiece);
PrevConvI.recv_cmd := false;
END_ACTION

ACTION Warehouse_Rst_Piece:
GVL.Reg[Roff] := 0;
END_ACTION

END_FUNCTION_BLOCK

// Device/Application/WarehouseIn_Conveyor
FUNCTION_BLOCK WarehouseIn_Conveyor
VAR_INPUT
	PrevConvI: Conv2Conv_fwd_T;
END_VAR
VAR_OUTPUT
	PrevconvO: Conv2Conv_bwd_T;
END_VAR
VAR
	Workpiece: Workpiece_T;
	Ioff: INT;
	Qoff: INT;
	Roff: INT;
END_VAR

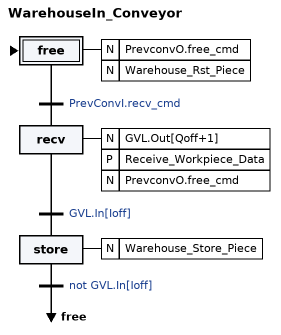
INITIAL_STEP free:
    PrevconvO.free_cmd(N);
    Warehouse_Rst_Piece(N);
END_STEP
TRANSITION FROM free TO recv
    := PrevConvI.recv_cmd;
END_TRANSITION
STEP recv:
    GVL.Out[Qoff+1](N);
    Receive_Workpiece_Data(P);
    PrevconvO.free_cmd(N);
END_STEP
TRANSITION FROM recv TO store
    := GVL.In[Ioff];
END_TRANSITION
STEP store:
    Warehouse_Store_Piece(N);
END_STEP
TRANSITION FROM store TO free
    := not GVL.In[Ioff];
END_TRANSITION

ACTION Warehouse_Store_Piece:
IF Qoff = 24 THEN
	GVL.Out[Qoff+3] := TRUE; // AT1_in5
ELSE
	GVL.Out[Qoff+2] := TRUE;
END_IF;
END_ACTION

//FB_Init is always available implicitly and it is used primarily for initialization.
//The return value is not evaluated. For a specific influence, you can also declare the
//methods explicitly and provide additional code there with the standard initialization
//code. You can evaluate the return value.
METHOD FB_Init: BOOL
VAR_INPUT
    bInitRetains: BOOL; // TRUE: the retain variables are initialized (reset warm / reset cold)
    bInCopyCode: BOOL;  // TRUE: the instance will be copied to the copy code afterward (online change)   
	Ioff_	: INT;
	Qoff_	: INT;
	Roff_	: INT;	
END_VAR
	Ioff := Ioff_;
	Qoff := Qoff_;
	Roff := Roff_;
END_METHOD

ACTION Warehouse_Rst_Piece:
GVL.Out[Qoff+2] := False;
END_ACTION

ACTION Receive_Workpiece_Data:
Workpiece := PrevConvI.Workpiece;
END_ACTION

END_FUNCTION_BLOCK

// Device/Application/Transfer_Cell
FUNCTION_BLOCK Transfer_Cell
VAR_INPUT
	PrevConvI: Conv2Conv_fwd_T;
END_VAR
VAR_OUTPUT
	PrevconvO: Conv2Conv_bwd_T;
END_VAR
VAR
	Wout : WarehouseOut_Conveyor(0, 0, 0);
	T1   : Linear_Conveyor(0, 0, 0);
	T2	 : Linear_Conveyor(0, 0, 0);
	T3	 : Linear_Conveyor(0, 0, 0);
	T4	 : Linear_Conveyor(0, 0, 0);
	T5	 : Linear_Conveyor(0, 0, 0);
	Win  : WarehouseIn_Conveyor(0, 0, 0);
END_VAR

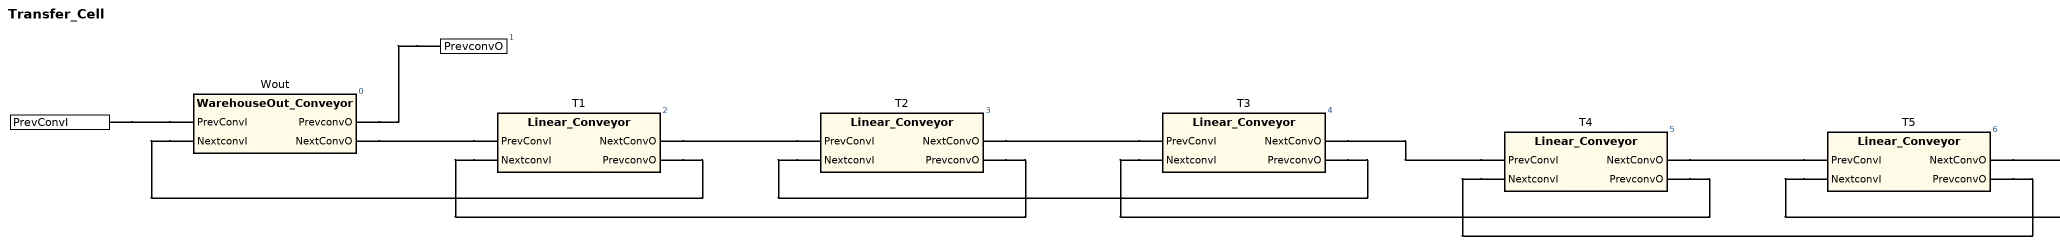
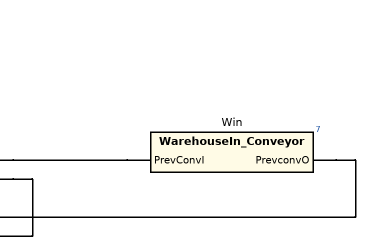
Wout(PrevConvI := PrevConvI, NextconvI := T1.PrevconvO); // WarehouseOut_Conveyor
PrevconvO := Wout.PrevconvO;
T1(PrevConvI := Wout.NextConvO, NextconvI := T2.PrevconvO); // Linear_Conveyor
T2(PrevConvI := T1.NextConvO, NextconvI := T3.PrevconvO); // Linear_Conveyor
T3(PrevConvI := T2.NextConvO, NextconvI := T4.PrevconvO); // Linear_Conveyor
T4(PrevConvI := T3.NextConvO, NextconvI := T5.PrevconvO); // Linear_Conveyor
T5(PrevConvI := T4.NextConvO, NextconvI := Win.PrevconvO); // Linear_Conveyor
Win(PrevConvI := T5.NextConvO); // WarehouseIn_Conveyor

//FB_Init is always available implicitly and it is used primarily for initialization.
//The return value is not evaluated. For a specific influence, you can also declare the
//methods explicitly and provide additional code there with the standard initialization
//code. You can evaluate the return value.
METHOD FB_Init: BOOL
VAR_INPUT
    bInitRetains: BOOL; // TRUE: the retain variables are initialized (reset warm / reset cold)
    bInCopyCode: BOOL;  // TRUE: the instance will be copied to the copy code afterward (online change) 
	Wout_I_ : INT; Wout_Q_ : INT; Wout_R_ : INT;
	T1_I_ : INT; T1_Q_ : INT;
	T2_I_ : INT; T2_Q_ : INT;
	T3_I_ : INT; T3_Q_ : INT;
	T4_I_ : INT; T4_Q_ : INT;
	T5_I_ : INT; T5_Q_ : INT;
	Win_I_ : INT; Win_Q_ : INT; Win_R_ : INT;  
END_VAR
	Wout.FB_Init(FALSE, FALSE, Wout_I_, Wout_Q_, Wout_R_);
	T1.FB_Init(FALSE, FALSE, T1_I_, T1_Q_, 0);
	T2.FB_Init(FALSE, FALSE, T2_I_, T2_Q_, 0);
	T3.FB_Init(FALSE, FALSE, T3_I_, T3_Q_, 0);
	T4.FB_Init(FALSE, FALSE, T4_I_, T4_Q_, 0);
	T5.FB_Init(FALSE, FALSE, T5_I_, T5_Q_, 0);
	Win.FB_Init(FALSE, FALSE, Win_I_, Win_Q_, Win_R_);
END_METHOD

END_FUNCTION_BLOCK

// Device/Application/SCADA_PRG
PROGRAM SCADA_PRG
VAR
END_VAR

Gate0 := GVL.Out[1];
Gate1 := GVL.Out[3];
Gate2 := GVL.Out[5];
S_sensor1 := GVL.In[0];
S_sensor2 := GVL.In[1];
S_sensor3 := GVL.In[2];
GVL.Out[1] := GVL.Out[1] AND (NOT C1_stop);
GVL.Out[3] := GVL.Out[3] AND (NOT C2_stop);
GVL.Out[5] := GVL.Out[5] AND (NOT C3_stop);

END_PROGRAM

// Device/Application/PRG_Loader
PROGRAM PRG_Loader
VAR
    Loader      : fb_Loader;
    i           : INT;

    // AT1_in0..4: Sensor I=5..9, Motor + at Q=10,13,16,19,22 (so WhIn pulse at Qoff+2)
    fb_WH_In0   : WarehouseIn_Conveyor( 5, 10, 0);
    fb_WH_In1   : WarehouseIn_Conveyor( 6, 13, 0);
    fb_WH_In2   : WarehouseIn_Conveyor( 7, 16, 0);
    fb_WH_In3   : WarehouseIn_Conveyor( 8, 19, 0);
    fb_WH_In4   : WarehouseIn_Conveyor( 9, 22, 0);

    aConvData   : ARRAY[0..4] OF Conv2Conv_fwd_T;

    // Cin0..Cin4 end-of-lane sensors
    cfg_Sensors           : ARRAY[0..4] OF INT := [0, 1, 2, 3, 4];
    // Cin0..Cin4 Motor − (feeds piece INTO the factory toward AT1_in)
    cfg_Motors            : ARRAY[0..4] OF INT := [1, 3, 5, 7, 9];
    // R Warehouse Out registers
    cfg_Spawns            : ARRAY[0..4] OF INT := [0, 1, 2, 3, 4];
    // AT1_in0..AT1_in4 sensors
    cfg_Sensors_Warehouse : ARRAY[0..4] OF INT := [5, 6, 7, 8, 9];
END_VAR

Loader(
    bExecute             := GVL.g_Loader_Exec,
    iTargetWood          := GVL.g_Loader_Wood_Qty,
    iTargetMetal         := GVL.g_Loader_Metal_Qty,
    aIn_Sensor           := cfg_Sensors,
    aOut_Motor           := cfg_Motors,
    aReg_Spawn           := cfg_Spawns,
    aIn_Sensor_Warehouse := cfg_Sensors_Warehouse   // was missing before
);

FOR i := 0 TO 4 DO
    aConvData[i].recv_cmd := (Loader.LaneState[i] >= 2);
END_FOR

fb_WH_In0(PrevConvI := aConvData[0]);
fb_WH_In1(PrevConvI := aConvData[1]);
fb_WH_In2(PrevConvI := aConvData[2]);
fb_WH_In3(PrevConvI := aConvData[3]);
fb_WH_In4(PrevConvI := aConvData[4]);

GVL.g_Loader_Status := Loader.iStatus;

END_PROGRAM

// Device/Application/fb_Loader
FUNCTION_BLOCK fb_Loader
VAR_INPUT
    bExecute      : BOOL;
    iTargetWood   : INT;
    iTargetMetal  : INT;
    // I/O offsets from io.csv — one entry per lane (0..4)
    aIn_Sensor  : ARRAY[0..4] OF INT;   // GVL.In  index for end-of-lane sensor
    aOut_Motor  : ARRAY[0..4] OF INT;   // GVL.Out index for lane motor
    aReg_Spawn  : ARRAY[0..4] OF INT;   // GVL.Reg index to spawn a piece
	
	aIn_Sensor_Warehouse : ARRAY[0..4] OF INT;	
END_VAR
VAR_OUTPUT
    iStatus : INT;   // 0=IDLE 1=LOADING 2=DONE 3=ERROR
END_VAR
VAR
    WoodSpawned   : INT := 0;
    MetalSpawned  : INT := 0;
    LaneState     : ARRAY[0..4] OF INT;
    i             : INT;
    rtExecute     : R_TRIG;
    AllLanesClear : BOOL;
    WOOD_ID       : UINT := 1;
    METAL_ID      : UINT := 2;
    // AT1_in Motor − addresses (pulls piece into the warehouse-in lane)
    aWHMotorMinus : ARRAY[0..4] OF INT := [11, 14, 17, 20, 23];
END_VAR

rtExecute(CLK := bExecute);

IF rtExecute.Q THEN
    WoodSpawned  := 0;
    MetalSpawned := 0;
    FOR i := 0 TO 4 DO
        LaneState[i]               := 0;
        GVL.Out[aOut_Motor[i]]     := FALSE;
        GVL.Out[aWHMotorMinus[i]]  := FALSE;
        GVL.Reg[aReg_Spawn[i]]     := 0;
    END_FOR
    iStatus := 1;
END_IF

IF iStatus = 1 THEN
    AllLanesClear := TRUE;
    FOR i := 0 TO 4 DO
        CASE LaneState[i] OF

            0:  // Idle: spawn next piece if Cin lane sensor is clear
                IF (WoodSpawned < iTargetWood) OR (MetalSpawned < iTargetMetal) THEN
                    IF NOT GVL.In[aIn_Sensor[i]] THEN
                        IF WoodSpawned < iTargetWood THEN
                            GVL.Reg[aReg_Spawn[i]] := WOOD_ID;
                            WoodSpawned := WoodSpawned + 1;
                        ELSE
                            GVL.Reg[aReg_Spawn[i]] := METAL_ID;
                            MetalSpawned := MetalSpawned + 1;
                        END_IF;
                        // Start Cin conveyor toward the factory floor (Motor −)
                        GVL.Out[aOut_Motor[i]] := TRUE;
                        LaneState[i] := 1;
                        AllLanesClear := FALSE;
                    END_IF
                END_IF

            1:  // Piece travelling on Cin, wait for Cin end-sensor to confirm arrival
                AllLanesClear := FALSE;
                IF GVL.In[aIn_Sensor[i]] THEN
                    // Piece reached end of Cin — start the AT1_in motor to pull it inward.
                    // Keep Cin motor running so the piece transitions onto AT1_in.
                    GVL.Out[aWHMotorMinus[i]] := TRUE;
                    LaneState[i] := 2;
                END_IF

            2:  // Wait for the AT1_in lane sensor to confirm the piece is on it
                AllLanesClear := FALSE;
                IF GVL.In[aIn_Sensor_Warehouse[i]] THEN
                    // Piece is on the warehouse-in lane → safe to stop the Cin belt
                    GVL.Out[aOut_Motor[i]] := FALSE;
                    GVL.Reg[aReg_Spawn[i]] := 0;
                    LaneState[i] := 3;
                END_IF

            3:  // Wait until AT1_in sensor clears (piece consumed by Warehouse-In FB)
                AllLanesClear := FALSE;
                IF NOT GVL.In[aIn_Sensor_Warehouse[i]] THEN
                    GVL.Out[aWHMotorMinus[i]] := FALSE;
                    LaneState[i] := 0;   // lane free for next piece
                END_IF

        END_CASE
    END_FOR

    IF (WoodSpawned >= iTargetWood) AND (MetalSpawned >= iTargetMetal) AND AllLanesClear THEN
        iStatus := 2;
    END_IF
END_IF

IF (NOT bExecute) AND (iStatus = 2) THEN
    iStatus := 0;
END_IF

END_FUNCTION_BLOCK

// Device/Application/Order_generator
PROGRAM Order_generator
VAR
    TransferTestCmd : INT := 0;
    TransferPiece : Workpiece_T;
END_VAR

GVL.Transfer_Order.recv_cmd := FALSE;

// Peça a transferir W2 -> W1
TransferPiece.InitPiece := 5; // exemplo: LegW
TransferPiece.Next_Operation := 0;
TransferPiece.Last_Operation := 0;

// Não precisa de operations reais porque não há machines.
// Mas preenche para manter a estrutura válida.
TransferPiece.Operations[0].Cell := 0;
TransferPiece.Operations[0].Machine := 0;
TransferPiece.Operations[0].Tool := 0;
TransferPiece.Operations[0].OpTime := T#0S;

CASE TransferTestCmd OF

1:
    GVL.Transfer_Order.Workpiece := TransferPiece;
    GVL.Transfer_Order.recv_cmd := TRUE;
    TransferTestCmd := 2;

2:
    GVL.Transfer_Order.recv_cmd := FALSE;

END_CASE

END_PROGRAM
